TYPE ST_GripperProcessConfig :
STRUCT
    tAcceptTimeout : TIME;
    tResultTimeout : TIME;
END_STRUCT
END_TYPE

(* stored: Version 1.1.0.1, ProductVersion 3.1.4026.20
   DUT ST_GripperProcessConfig: Id {d30a5618-339b-4dcc-a09f-71dec6b142dc} *)
